FUNCTION_BLOCK "EM_Heating"
{ S7_Optimized_Access := 'TRUE' }
BEGIN
// No networks contain logic in the TIA project
END_FUNCTION_BLOCK
